FUNCTION_BLOCK FB_exitConveyorTrigger
VAR_INPUT
	inputLeft : BOOL;
	inputRight : BOOL;
	inputForward : BOOL;
END_VAR
VAR_OUTPUT
	leftEdge : BOOL;
	rightEdge : BOOL;
	frontEdge : BOOL;
END_VAR
VAR
	rTrigLeft : Tc2_Standard.R_TRIG;
	rTrigRight : Tc2_Standard.R_TRIG;
	rTrigForward : Tc2_Standard.R_TRIG;
END_VAR

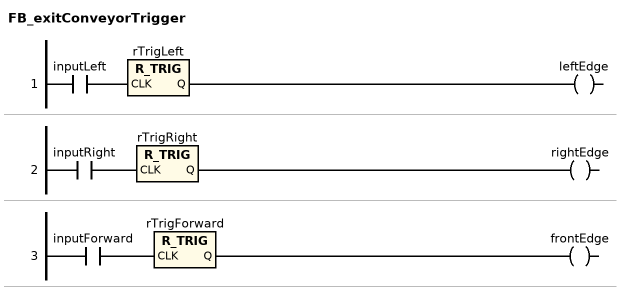
// NETWORK 1
rTrigLeft(CLK := inputLeft); // R_TRIG
leftEdge := rTrigLeft.Q;

// NETWORK 2
rTrigRight(CLK := inputRight); // R_TRIG
rightEdge := rTrigRight.Q;

// NETWORK 3
rTrigForward(CLK := inputForward); // R_TRIG
frontEdge := rTrigForward.Q;

END_FUNCTION_BLOCK

(* stored: Version 1.1.0.1, ProductVersion 3.1.4024.13
   POU FB_exitConveyorTrigger: Id {a84237e8-0ba1-4c68-93e5-98d8d1726c6e}, SpecialFunc None *)
